SUBAPPLICATION Softkey_Aux_Switch_TO_Remote_WRITE (* VT-SoftKey lesen ODER AUX-Zuweisung (Joystick) lesen ODER lokaler Web-Override (z.B. vt-ui-mirror auf demselben Modul) ODER ein zusaetzlicher physischer Taster auf einem ANDEREN Modul (Remote-Subscribe) + Remote-OPC-UA-Write an Zielmodul (generisch, ein Kanal, ohne Status-Feedback) - 4-Quellen-Erweiterung von Softkey_Aux_IXA_TO_Remote_WRITE fuer Funktionen, die zusaetzlich zu SoftKey/AUX/Web noch einen fest verbauten Taster auf einem dritten Modul haben (z.B. Schnittverstellung: SoftKey auf STG1, Taster S06/S07 auf STG4, Aktor auf STG2) *)
  (* Standard: 61499-2; Description: Copyright (c) 2026 Meisterschulen am Ostbahnhof This program and the accompanying materials are made available under the terms of the Eclipse Public License 2.0 which is available at https://www.eclipse.org/legal/epl-2.0/ SPDX-License-Identifier: EPL-2.0 *)
  (* Version 1.0, 2026-09-07, Franz Höpfinger, Meisterschulen am Ostbahnhof, initial API and implementation and/or initial documentation - 4-Quellen-Variante von Softkey_Aux_IXA_TO_Remote_WRITE fuer Schnittverstellung (V14: SoftKey_Aufnahme_Heben/Senken auf STG1, physische Taster S06/S07 auf STG4, Aktor auf STG2) *)
  PACKAGE MyLib::sys;
  IMPORT isobus::UT::Q::const::IDs::ID_NULL;
  (* Documentation:
  SoftKey UND Aux UND Web UND Remote-Taster → Remote-OPC-UA-Write (nur Kommando, kein Status)
   4-Quellen-Erweiterung von Softkey_Aux_IXA_TO_Remote_WRITE: zusaetzlich zu SoftKey (u16ObjId), Aux-Zuweisung (u16ObjIdA) und lokalem Web-Override (ID_WEB_READ) wird noch ein vierter, per Remote-Subscribe gelesener physischer Taster auf einem ANDEREN Modul (ID_SWITCH_REMOTE) per AX_OR_4 zusammengefuehrt und per AX_CLIENT_1_0 (ID_WRITE_REMOTE) ans Zielmodul geschrieben.
   Wichtig: alle 4 Quellen werden HIER (auf dem Bedienmodul, z.B. STG1) zu EINEM Kommando zusammengefuehrt, bevor per EINEM einzigen AX_CLIENT_1_0 ans Zielmodul geschrieben wird - NICHT mehrere unabhaengige Writer auf denselben Zielknoten (das waere ein Race/Last- Write-Wins-Fehler, kein echtes ODER). Fuer den Anwendungsfall Schnittverstellung: SoftKey_ Aufnahme_Heben/Senken (STG1) + AuxFunction2 (Joystick) + vt-ui-mirror-Web-Override, ALLE auf STG1, ODER-verknuepft mit dem physischen Taster S06/S07 (STG4, per Remote-Subscribe STG4_I2/ I3_REMOTE - bereits fuer die VT-IO-Diag-Anzeige vorhanden, hier zusaetzlich mitverwendet).
   Kein Status-Feedback/Hintergrundfarbe hier - dafuer AX_SUBSCRIBE_BG3_WEB_OPC danebenstellen (gleiche u16ObjId/u16ObjIdA-Werte durchreichen), genau wie bei Softkey_Aux_IXA_TO_Remote_WRITE.
  *)
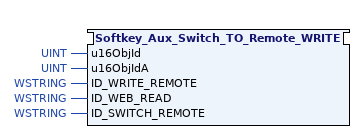
  VAR_INPUT
    u16ObjId : UINT := ID_NULL; (* Object ID SoftKey (VT) *)
    u16ObjIdA : UINT := ID_NULL; (* Object ID AuxFunction2 (VT) *)
    ID_WRITE_REMOTE : WSTRING; (* Remote-Write-Adresse zum Zielmodul (Befehl, ACTION=WRITE, CLIENT) *)
    ID_WEB_READ : WSTRING; (* Lokale Subscribe-Adresse fuer einen Web-Client (z.B. vt-ui-mirror) auf demselben Modul, ODER-verknuepft mit SoftKey und AUX *)
    ID_SWITCH_REMOTE : WSTRING; (* Remote-Subscribe-Adresse eines zusaetzlichen physischen Tasters auf einem ANDEREN Modul (z.B. STG4_I2_REMOTE), ODER-verknuepft mit SoftKey/AUX/Web *)
  END_VAR
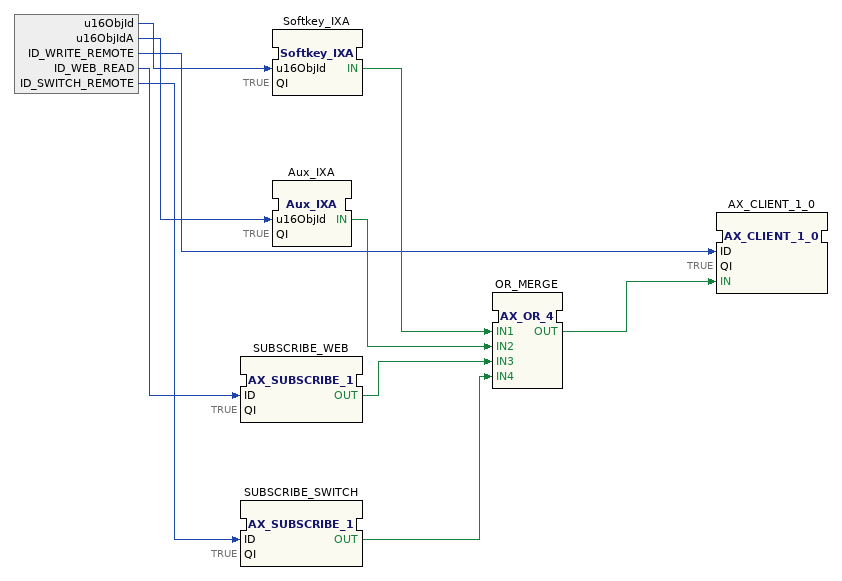
  FBS
    Softkey_IXA : isobus::UT::io::Softkey::Softkey_IXA(QI := TRUE);
    Aux_IXA : isobus::UT::io::Auxiliary::IN::Aux_IXA(QI := TRUE);
    SUBSCRIBE_WEB : adapter::net::AX_SUBSCRIBE_1(QI := TRUE);
    SUBSCRIBE_SWITCH : adapter::net::AX_SUBSCRIBE_1(QI := TRUE);
    OR_MERGE : adapter::booleanOperators::AX_OR_4;
    AX_CLIENT_1_0 : adapter::net::AX_CLIENT_1_0(QI := TRUE);
  END_FBS
  DATA_CONNECTIONS
    u16ObjId TO Softkey_IXA.u16ObjId;
    u16ObjIdA TO Aux_IXA.u16ObjId;
    ID_WEB_READ TO SUBSCRIBE_WEB.ID;
    ID_SWITCH_REMOTE TO SUBSCRIBE_SWITCH.ID;
    ID_WRITE_REMOTE TO AX_CLIENT_1_0.ID;
  END_CONNECTIONS
  ADAPTER_CONNECTIONS
    Softkey_IXA.IN TO OR_MERGE.IN1;
    Aux_IXA.IN TO OR_MERGE.IN2;
    SUBSCRIBE_WEB.OUT TO OR_MERGE.IN3;
    SUBSCRIBE_SWITCH.OUT TO OR_MERGE.IN4;
    OR_MERGE.OUT TO AX_CLIENT_1_0.IN;
  END_CONNECTIONS
END_SUBAPPLICATION
